RoboDK station: Stringer A - Top Down - BOX1.rdk

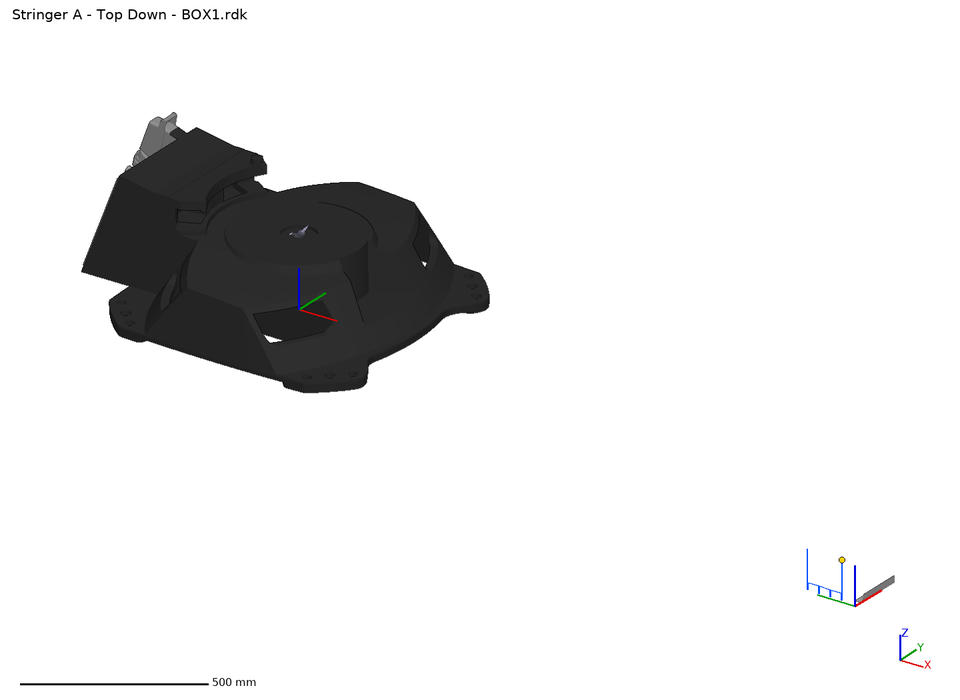
[picture v0: the station drawn from its stored meshes, robots at their saved joint values, targets as dots, program paths as lines]
Station Stringer A - Top Down - BOX1 (saved by RoboDK 5.2.3). Poses are relative to the parent item; angles as X-Y-Z fixed-axis rotations.
  - frame KUKA KR 210 R2700 extra Base at (0, 0, 0) mm
    - robot KUKA KR 210 R2700 extra: 6 axes, payload 210 kg, reach 2696 mm, repeatability 0.06 mm, weight 1068 kg
        joint limits [-185, -140, -120, -350, -125, -350] to [185, -5, 155, 350, 125, 350]; home [0, -90, 90, 0, 0, 0]; saved at [-6.051, -33.956, 111.537, 171.503, 26.677, -177.106]
      - tool Spindle, TCP at (32, 0, 260) mm, rotated rx 0 ry 39 rz 0 deg, size 157.3 x 72 x 259.9 mm
  - frame Frame 2 at (1800, 0, -372.68) mm, rotated rx 0 ry 0 rz 90 deg
    - object Stringer A-TopDOWN-BOX1 at (0, 22.5, 0) mm, rotated rx 0 ry 0 rz -90 deg, 4 curves, geometry from Point 4
    - object L-Stringer A - top down at (0, 0, 0) mm, size 151.7 x 20 x 20 mm, geometry from L-Stringer A - top down.stl
  - machining project Point settings: rotZ(0) | rotX(0)*rotY(0) | rotz(0) | onStart | onPathStart | onApproach | onPoint | onRetract | onFinish | SetRPM(%1) | SetTool(%1) | Extruder(%1) | default | default | OutOnMov(%1) | OutOffMov(%1) | onPathFinish | M_RunCode(%1)
  - program Point (31 instructions, listed below)
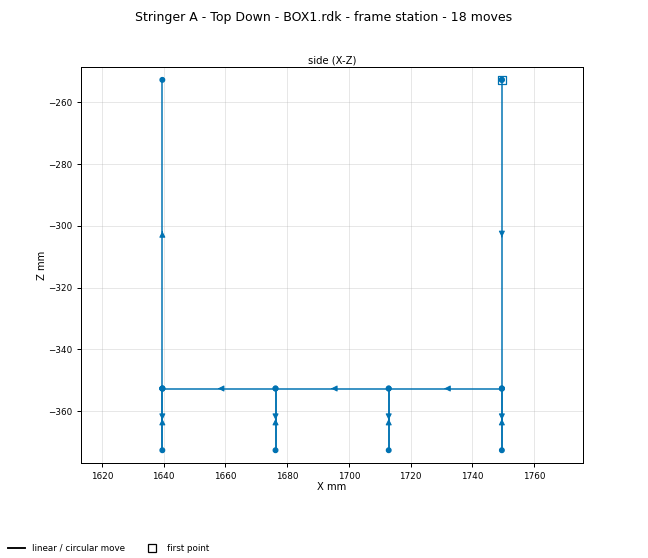
[picture p0: tool path of Stringer A - Top Down - BOX1.rdk in frame station, 18 of 18 moves have a stored position in this frame; points joined in program order, loops and branches not executed]

--- program Point (robot KUKA KR 210 R2700 extra) ---
  Smooth(1)
  Set speed (1000.0 mm/s)
  Set Ref.: Frame 2
  Set Tool: Spindle
  Show Spindle
  MoveJ 1 to (10, 50.43, 120) mm, rotated rx 180 ry 0 rz 180 deg; joints [-1.908, -34.03, 111.941, 177.347, 26.92, -179.117]
  MoveL 2 to (10, 50.43, 120) mm, rotated rx 180 ry 0 rz 180 deg; joints [-1.908, -34.03, 111.941, 177.347, 26.92, -179.117]
  MoveL 3 to (10, 50.43, 20) mm, rotated rx -180 ry 0 rz -180 deg; joints [-1.908, -28.696, 109.297, 177.569, 29.607, -179.369]
  MoveL 4 to (10, 50.43, 20) mm, rotated rx -180 ry 0 rz -180 deg; joints [-1.908, -28.696, 109.297, 177.569, 29.607, -179.369]
  Set speed (50.0 mm/s)
  MoveL 5 to (10, 50.43, 0) mm, rotated rx 180 ry 0 rz -180 deg; joints [-1.908, -27.637, 108.721, 177.604, 30.089, -179.41]
  MoveL 6 to (10, 50.43, 20) mm, rotated rx -180 ry 0 rz -180 deg; joints [-1.908, -28.696, 109.297, 177.569, 29.607, -179.369]
  Set speed (1000.0 mm/s)
  MoveL 7 to (10, 87.09, 20) mm, rotated rx 180 ry 0 rz -180 deg; joints [-3.293, -28.684, 109.211, 175.795, 29.546, -178.901]
  Set speed (50.0 mm/s)
  MoveL 8 to (10, 87.09, 0) mm, rotated rx 180 ry 0 rz 180 deg; joints [-3.293, -27.626, 108.635, 175.857, 30.027, -178.972]
  MoveL 9 to (10, 87.09, 20) mm, rotated rx 180 ry 0 rz -180 deg; joints [-3.293, -28.684, 109.211, 175.795, 29.546, -178.901]
  Set speed (1000.0 mm/s)
  MoveL 10 to (10, 123.76, 20) mm, rotated rx 180 ry 0 rz 180 deg; joints [-4.675, -28.666, 109.078, 174.012, 29.452, -178.418]
  Set speed (50.0 mm/s)
  MoveL 11 to (10, 123.76, 0) mm, rotated rx -180 ry 0 rz -180 deg; joints [-4.675, -27.61, 108.503, 174.1, 29.931, -178.519]
  MoveL 12 to (10, 123.76, 20) mm, rotated rx 180 ry 0 rz 180 deg; joints [-4.675, -28.666, 109.078, 174.012, 29.452, -178.418]
  Set speed (1000.0 mm/s)
  MoveL 13 to (10, 160.43, 20) mm, rotated rx -180 ry 0 rz -180 deg; joints [-6.051, -28.642, 108.9, 172.216, 29.328, -177.913]
  Set speed (50.0 mm/s)
  MoveL 14 to (10, 160.43, 0) mm, rotated rx 180 ry 0 rz -180 deg; joints [-6.051, -27.587, 108.325, 172.33, 29.804, -178.044]
  MoveL 15 to (10, 160.43, 20) mm, rotated rx -180 ry 0 rz -180 deg; joints [-6.051, -28.642, 108.9, 172.216, 29.328, -177.913]
  MoveL 16 to (10, 160.43, 20) mm, rotated rx -180 ry 0 rz -180 deg; joints [-6.051, -28.642, 108.9, 172.216, 29.328, -177.913]
  Set speed (1000.0 mm/s)
  MoveL 17 to (10, 160.43, 20) mm, rotated rx -180 ry 0 rz -180 deg; joints [-6.051, -28.642, 108.9, 172.216, 29.328, -177.913]
  MoveL 18 to (10, 160.43, 120) mm, rotated rx -180 ry 0 rz -180 deg; joints [-6.051, -33.956, 111.537, 171.503, 26.677, -177.106]
